# EPICS substitutions: TagApp/Db/notifyString.substitutions
file "notifyString.template" {

# PV name is $(Sys)$(Dev)$(Attr)

# UUID selects the sensor to be read; must be notify type
#	Note that EPICS doesn't like a leading zero, so the first zero is omitted
# http://processors.wiki.ti.com/index.php/CC2650_SensorTag_User's_Guide

pattern { Sys, 	Dev  		  ,	Attr 		 ,		UUID}

}
